{attribute 'GeneratedUsingTerminal: AES-D-BC-ECAT Gen2-0001'}
{attribute addProperty BoxType "AES-D-BC-ECAT Gen2-0001"}
{attribute addProperty Id "Web_App_DisableAT %Q*BOOL1Freeze_OutputAT %Q*BOOL1HL_SwapAT %Q*BOOL1Default_Modul_ControlAT %Q*BOOL1"}
{attribute addProperty CRC "1649935978"}
{attribute addProperty Size "4"}
TYPE Device_Control_6258066A EXTENDS TcoIo.OutputBase_10CEE7DE :
STRUCT
	{attribute addProperty Name "Web_App_Disable"}
	Web_App_Disable AT %Q* : BOOL;
	{attribute addProperty Name "Freeze_Output"}
	Freeze_Output AT %Q* : BOOL;
	{attribute addProperty Name "HL_Swap"}
	HL_Swap AT %Q* : BOOL;
	{attribute addProperty Name "Default_Modul_Control"}
	Default_Modul_Control AT %Q* : BOOL;
END_STRUCT
END_TYPE

(* stored: Version 1.2.0.0, ProductVersion 3.1.4024.9
   DUT Device_Control_6258066A: Id {a307a5ce-9452-09d5-3b35-e09896b58ccc} *)
